(* CoDeSys 2.3.9.37 project: Cap8_4.pro *)
(* Libraries: Standard.lib 4.10.05 12:14:46 *)

(* Global variable list: Global_Variables *)
VAR_GLOBAL

    (* Entradas *)
     Interruptor:BOOL;
     FuncNormal:BOOL;

     (* Salidas *)
     RojoCoche:BOOL;
     AmbarCoche:BOOL;
    VerdeCoche:BOOL;
    RojoPeaton:BOOL;
     VerdePeaton:BOOL;
END_VAR

(* POU PLC_PRG, IL *)
PROGRAM PLC_PRG
VAR
END_VAR

END_PROGRAM

(* Visualisation Visu
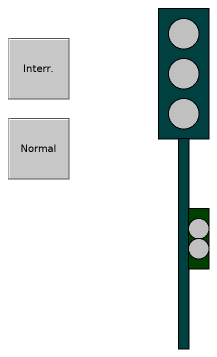
button at (20,50)-(81,111): text "Interr."; toggles Interruptor
button at (20,130)-(81,191): text "Normal"; toggles FuncNormal
ellipse at (180,30)-(211,61): alarm colour if RojoCoche
ellipse at (180,70)-(211,101): alarm colour if AmbarCoche
ellipse at (180,110)-(211,141): alarm colour if VerdeCoche
ellipse at (200,230)-(221,251): alarm colour if RojoPeaton
ellipse at (200,250)-(221,271): alarm colour if VerdePeaton
3 more shapes without text or variables
*)
